# EPICS autosave request: mrfApp/Db/evr-common.inc.req
$(P)$(R)DBus:SharedRX.VAL
$(P)$(R)DBus:SharedTX.VAL
$(P)$(R)DataBuffer:TX:Enabled.VAL
$(P)$(R)DataBuffer:TX:TransferSize.VAL
$(P)$(R)DataBuffer:TX:TransmitData.VAL
$(P)$(R)Enabled.VAL
$(P)$(R)Event:Log:StopEventEnabled.VAL
$(P)$(R)Event:MapRAM:Enabled.VAL
$(P)$(R)Event:MapRAM:Select.VAL
$(P)$(R)EventClock:Freq.VAL
$(P)$(R)EventClock:Gen:Freq.VAL
$(P)$(R)RX:Loopback.VAL
$(P)$(R)TX:Loopback.VAL
$(P)$(R)TimeStamp:EventCounterPrescaler.VAL
$(P)$(R)TimeStamp:EventCounterSource.VAL
